	            IF #Transf.Dial_Def.Reponse_Def = 'Cellule' AND #Transf.Dial_Def.Num_Def_Etape = 1 THEN // cellule
	                #Ret_Int := "Index_Mobile"(#Transf.Dial_Def.Text_Reponse);
	                #Transf.Dial_Def.Reponse_Def := '';
	                IF #Ret_Int <= -1 THEN
	                    #Text_Def := CONCAT(IN1 := 'Cellule ', IN2 := #Transf.Dial_Def.Text_Reponse, IN3 := ' Inexistante');
	                    #Transf.Dial_Def.Index_Defaut := "Dialog_Defaut"(Fg_Base := #fgbase, Msg_Defaut := #Text_Def,
	                                                                     Type_Defaut := 2,
	                                                                     Automatisme := #Transf._TransfCommun.CommunGeneral._Autom,
	                                                                     Num_Lot := #Transf._PtCir.Num_Lot,
	                                                                     Origine_Defaut := #Text_Def,
	                                                                     Libelle_Origine := 'Cellule inexistante',
	                                                                     Acq1 := 'Relance',
	                                                                     Acq2 := 'Cellule',
	                                                                     Acq3 := '',
	                                                                     Acq4 := '',
	                                                                     Acq5 := '',
	                                                                     Acq6 := '',
	                                                                     Acq7 := '',
	                                                                     Acq8 := '',
	                                                                     Acq_Choisi := -1,
	                                                                     Date_Arrivee := #Transf._TpsPicke);
	                    #Transf._TransfCommun.CommunGeneral._Etp := #Etape_Attente_RepDial;
	                    #Transf.Dial_Def.Text_Reponse := '';
	                    RETURN;
	                ELSE
	                    #Transf._CelluleTrouve := "Controle_Cellule"(FgMaskNh := #Transf._FgMaskCtrlNh,
	                                                                 NvCellule := #Transf.Dial_Def.Text_Reponse,
	                                                                 TypeCelDest := #Transf._TypeCelDest,
	                                                                 Cel := "DB_Mod_Cellule",
	                                                                 NiveauHautDestNh => #Transf._NiveauHautDestNh);
	                END_IF;
	            END_IF;
	            //============ fIN Traitement des reponses pour le defaut1 Etape CHANGEMENT DE DESTINATION cellule introuvable  ===============================//






	            ////Test invalide de la destination recuperee de la Base, cellule est en nh
	            IF #Transf._CelluleTrouve = 1 THEN
	                #Transf.Dial_Def.Num_Def_Etape := 2;
	                #Text_Def := CONCAT(IN1 := 'Cellule ', IN2 := #Transf.Dial_Def.Text_Reponse, IN3 := '  est en NH');
	                #Transf.Dial_Def.Index_Defaut := "Dialog_Defaut"(Fg_Base := #fgbase, Msg_Defaut := #Text_Def,
	                                                                 Type_Defaut := 2,
	                                                                 Automatisme := #Transf._TransfCommun.CommunGeneral._Autom,
	                                                                 Num_Lot := #Transf._Ptzs._NoLot,
	                                                                 Origine_Defaut := #Text_Def,
	                                                                 Libelle_Origine := #Text_Def,
	                                                                 Acq1 := 'Relance',
	                                                                 Acq2 := 'Cellule',
	                                                                 Acq3 := '', //'Forçage'
	                                                                 Acq4 := '',
	                                                                 Acq5 := '',
	                                                                 Acq6 := '',
	                                                                 Acq7 := '',
	                                                                 Acq8 := '',
	                                                                 Acq_Choisi := -1,
	                                                                 Date_Arrivee := #Transf._TpsPicke);
	                #Transf._TransfCommun.CommunGeneral._Etp := #Etape_Attente_RepDial;
	                RETURN;
	            END_IF;
	        CHANGEMENT_DEST_DEF2:
	            //============ Traitement des reponses pour le defaut2 Etape CHANGEMENT DE DESTINATION cellule en nh  ====================================//
	            IF #Transf.Dial_Def.Reponse_Def = 'Relance' AND #Transf.Dial_Def.Num_Def_Etape = 2 THEN
	                #Transf._CelluleTrouve := "Controle_Cellule"(FgMaskNh := #Transf._FgMaskCtrlNh,
	                                                             NvCellule := #Transf.Dial_Def.Text_Reponse,
	                                                             TypeCelDest := #Transf._TypeCelDest,
	                                                             Cel := "DB_Mod_Cellule",
	                                                             NiveauHautDestNh => #Transf._NiveauHautDestNh);
	                #Transf.Dial_Def.Text_Reponse := '';
	                RETURN;
	            END_IF;


	            IF #Transf.Dial_Def.Reponse_Def = 'Forcage' AND #Transf.Dial_Def.Num_Def_Etape = 2 THEN
	                #Transf._FgMaskCtrlNh := TRUE;
	                #Transf._FgChangDest := FALSE;
	                #Transf._TransfCommun.SUPTRANS.Commande._FgChangDest := FALSE;
	                #Transf._Ptzs._DestR._Liste[#Transf._Ptzs._DestR._Index]._Nh := FALSE;
	                #Transf._CelluleTrouve := 2;
	                #Transf._TransfCommun.CommunGeneral._Ptdest := "Index_Mobile"(#Transf.Dial_Def.Text_Reponse);
	                #Transf._IndexDestEc := "RechIndexCel"("Nom_Mobile"(#Transf._TransfCommun.CommunGeneral._Ptdest));
	                IF #Transf._IndexDestEc > -1 THEN
	                    #Transf._ptDestEc := "DB_Mod_Cellule"._TabCel[#Transf._IndexDestEc];
	                END_IF;
	                (* "MAJ_Cumul_Dest"(Dest := "Nom_Mobile"(#Transf.TransfCommun.CommunGeneral._Ptdest),
	                                  Increment := FALSE,
	                                  DestR := #Transf._Ptzs._DestR,
	                                  PARCAL := #Transf.TransfCommun.CommunGeneral._ParCal);
	                 #Transf._CumulQteNh := #Transf._Ptzs._DestR._Liste[#Transf._Ptzs._DestR._Index]._CumulQte;
	                 (* #Transf.transfCommun.CommunGeneral._Ptdest := "Index_Mobile"(#Transf.Dial_Def.Text_Reponse);
	                 #Transf._IndexDestEc := "RechIndexCel"("Nom_Mobile"(#Transf.transfCommun.CommunGeneral._Ptdest)); *)
	                "ChngDestNoeud_Transfert"(#Transf); *)
	                #Transf.Dial_Def.Reponse_Def := '';
	            END_IF;



	            IF #Transf.Dial_Def.Reponse_Def = 'Cellule' AND #Transf.Dial_Def.Num_Def_Etape = 2 THEN // cellule
	                #Ret_Int := "Index_Mobile"(#Transf.Dial_Def.Text_Reponse);
	                #Transf.Dial_Def.Reponse_Def := '';
	                IF #Ret_Int <= -1 THEN
	                    #Transf._CelluleTrouve := 0;
	                    #Transf.Dial_Def.Num_Def_Etape := 1;
	                    #Text_Def := CONCAT(IN1 := 'Cellule ', IN2 := #Transf.Dial_Def.Text_Reponse, IN3 := '  inexistante');
	                    #Transf.Dial_Def.Index_Defaut := "Dialog_Defaut"(Fg_Base := #fgbase, Msg_Defaut := #Text_Def,
	                                                                     Type_Defaut := 2,
	                                                                     Automatisme := #Transf._TransfCommun.CommunGeneral._Autom,
	                                                                     Num_Lot := #Transf._PtCir.Num_Lot,
	                                                                     Origine_Defaut := 'Cellule inexistante',
	                                                                     Libelle_Origine := 'Cellule inexistante',
	                                                                     Acq1 := 'Relance',
	                                                                     Acq2 := 'Cellule',
	                                                                     Acq3 := '',
	                                                                     Acq4 := '',
	                                                                     Acq5 := '',
	                                                                     Acq6 := '',
	                                                                     Acq7 := '',
	                                                                     Acq8 := '',
	                                                                     Acq_Choisi := -1,
	                                                                     Date_Arrivee := #Transf._TpsPicke);
	                    #Transf._TransfCommun.CommunGeneral._Etp := #Etape_Attente_RepDial;
	                    #Transf.Dial_Def.Text_Reponse := '';
	                    RETURN;
	                ELSE
	                    #Transf._CelluleTrouve := "Controle_Cellule"(FgMaskNh := #Transf._FgMaskCtrlNh,
	                                                                 NvCellule := #Transf.Dial_Def.Text_Reponse,
	                                                                 TypeCelDest := #Transf._TypeCelDest,
	                                                                 Cel := "DB_Mod_Cellule",
	                                                                 NiveauHautDestNh => #Transf._NiveauHautDestNh);
	                END_IF;
	            END_IF;

	            //============ FIN Traitement des reponses pour le defaut2 Etape CHANGEMENT DE DESTINATION cellule en nh  ====================================//



	            IF #Transf._CelluleTrouve = 3 THEN // CELLULE RECUP VALID MAIS LA RECHERCHERCHE DU NV CIRC RETURN-1
	                #Transf.Dial_Def.Num_Def_Etape := 1;
	                #Text_Def := CONCAT(IN1 := 'Circuit de ', IN2 := "Nom_Mobile"(#Transf._TransfCommun.CommunGeneral._PtOrig), IN3 := ' vers ', IN4 := #Transf.Dial_Def.Text_Reponse, IN5 := ' introuvable ou reserve ');
	                #Transf.Dial_Def.Index_Defaut := "Dialog_Defaut"(Fg_Base := #fgbase, Msg_Defaut := #Text_Def,
	                                                                 Type_Defaut := 2,
	                                                                 Automatisme := #Transf._TransfCommun.CommunGeneral._Autom,
	                                                                 Num_Lot := #Transf._Ptzs._NoLot,
	                                                                 Origine_Defaut := 'Circuit Introuvable',
	                                                                 Libelle_Origine := 'Circuit Introuvable',
	                                                                 Acq1 := 'Relance',
	                                                                 Acq2 := 'Cellule',
	                                                                 Acq3 := '',
	                                                                 Acq4 := '',
	                                                                 Acq5 := '',
	                                                                 Acq6 := '',
	                                                                 Acq7 := '',
	                                                                 Acq8 := '',
	                                                                 Acq_Choisi := -1,
	                                                                 Date_Arrivee := #Transf._TpsPicke);
	                #Transf._TransfCommun.CommunGeneral._Etp := #Etape_Attente_RepDial;
	                RETURN;
	            END_IF;


	            //Test valide de la destination recuperee
	            IF #Transf._CelluleTrouve = 2 THEN
	                IF #Transf._TransfCommun.CommunGeneral._IndxDest <> #ListeDestParcourue THEN
	                    #CdZoneDest := "Nom_Mobile"(#Transf._TransfCommun.CommunGeneral._Dest[#Transf._TransfCommun.CommunGeneral._IndxDest]);
	                ELSE
	                    #CdZoneDest := #Transf.Dial_Def.Text_Reponse;
	                END_IF;
	                #Anc_Dest := "Nom_Mobile"(#Transf._TransfCommun.CommunGeneral._AncDest);
	                (* "ControleDestTransf"(fgbase := fgbase,
	                                     "Return" => #Ret_Int,
	                                     Transf := #Transf,
	                                     NoLot := #Transf._Ptzs._NoLot,
	                                     CdZoneDest := #CdZoneDest,
	                                     Anc_Dest := #Anc_Dest,
	                                     Nouv_Dest := #Transf._Ptzs._NouvDest,
	                                     CdMat := #Transf._Ptzs._CdMat,
	                                     NomAuto := #Transf.TransfCommun.CommunGeneral._Autom); *)

	                "ControleDest"(fgbase := #fgbase,
	                               TypeCelDest := #Transf._TypeCelDest,
	                               FgMaskCtrlNh := #Transf._FgMaskCtrlNh,
	                               "Return" => #Ret_Int,
	                               FgLanc => #Transf._FgLanc,
	                               NiveauHautDestNh => #Transf._NiveauHautDestNh,
	                               CntlDest := #Transf.CntlDest,
	                               Dial_Def := #Transf.Dial_Def,
	                               NoLot := #Transf._Ptzs._NoLot,
	                               CdZoneDest := #CdZoneDest,
	                               Anc_Dest := #Anc_Dest,
	                               Nouv_Dest := #Transf._Ptzs._NouvDest,
	                               CdMat := #Transf._Ptzs._CdMat,
	                               NomAuto := #Transf._TransfCommun.CommunGeneral._Autom);

	                IF #Ret_Int = -1 THEN
	                    #Transf._CelluleTrouve := 0;
	                END_IF;
	                IF #Ret_Int = 1 THEN
	                    #Transf._CumulQteNh := #Transf._Ptzs._DestR._Liste[#Transf._Ptzs._DestR._Index]._CumulQte;
	                    // IF #Transf.TransfCommun.CommunGeneral._IndxDest <= "NB_MAX_DEST" THEN //AND #Transf.Dial_Def.Num_Def_Etape = 0 THEN
	                    IF #Transf._TransfCommun.CommunGeneral._IndxDest <> #ListeDestParcourue THEN
	                        #Transf._TransfCommun.CommunGeneral._Ptdest := #Transf._TransfCommun.CommunGeneral._Dest[#Transf._TransfCommun.CommunGeneral._IndxDest];
	                    ELSE
	                        #Transf._TransfCommun.CommunGeneral._Ptdest := "Index_Mobile"(#Transf.Dial_Def.Text_Reponse);
	                    END_IF;
	                    #Transf._IndexDestEc := "RechIndexCel"("Nom_Mobile"(#Transf.#_TransfCommun.CommunGeneral._Ptdest));
	                    IF #Transf._IndexDestEc > -1 THEN
	                        #Transf._ptDestEc := "DB_Mod_Cellule"._TabCel[#Transf._IndexDestEc];
	                    END_IF;
	                    #Transf._TransfCommun.CommunGeneral._Etp := #Etape_ChgmtDestNoeud;
	                    RETURN;

	                END_IF;


	                (* #Transf._CumulQteNh := #Transf._Ptzs._DestR._Liste[#Transf._Ptzs._DestR._Index]._CumulQte;
	                 // IF #Transf.TransfCommun.CommunGeneral._IndxDest <= "NB_MAX_DEST" THEN //AND #Transf.Dial_Def.Num_Def_Etape = 0 THEN
	                 IF #Transf.TransfCommun.CommunGeneral._IndxDest <> #ListeDestParcourue THEN
	                     #Transf.TransfCommun.CommunGeneral._Ptdest := #Transf.TransfCommun.CommunGeneral._Dest[#Transf.TransfCommun.CommunGeneral._IndxDest];
	                 ELSE
	                     #Transf.TransfCommun.CommunGeneral._Ptdest := "Index_Mobile"(#Transf.Dial_Def.Text_Reponse);
	                 END_IF;
	                 #Transf._IndexDestEc := "RechIndexCel"("Nom_Mobile"(#Transf.#TransfCommun.CommunGeneral._Ptdest));
	                 IF #Transf._IndexDestEc > -1 THEN
	                     #Transf._ptDestEc := "DB_Mod_Cellule"._TabCel[#Transf._IndexDestEc];
	                 END_IF;
	                 "ChngDestNoeud_Transfert"(#Transf); *)
	            END_IF;







	            (* IF #Transf.TransfCommun.CommunGeneral._IndxDest <> #ListeDestParcourue THEN
	                 #CdZoneDest := "Nom_Mobile"(#Transf.TransfCommun.CommunGeneral._Dest[#Transf.TransfCommun.CommunGeneral._IndxDest]);
	             ELSE
	                 #CdZoneDest := #Transf.Dial_Def.Text_Reponse;
	             END_IF;
	             #Anc_Dest := "Nom_Mobile"(#Transf.TransfCommun.CommunGeneral._AncDest);
	             "ControleDestTransf"(fgbase:=fgbase,
	                                  "Return"=>#Ret_Int,
	                                  Transf:=#Transf,
	                                  NoLot:=#Transf._Ptzs._NoLot,
	                                  CdZoneDest:= #CdZoneDest,
	                                  Anc_Dest:= #Anc_Dest,
	                                  Nouv_Dest:=#Transf._Ptzs._NouvDest,
	                                  CdMat:=#Transf._Ptzs._CdMat,
	                                  NomAuto:=#Transf.TransfCommun.CommunGeneral._Autom);
	             IF #Ret_Int =1 THEN
	                 #Transf._CelluleTrouve := 2 ;
	             ELSE
	                 #Transf._CelluleTrouve := -2;
	             END_IF; *)

	        END_REGION Traitement cyclique
	(*
	 *************************************** *************************************** *************************************** *************************************** *************************************** ***************************************
	                                                                                 ╔════════════════════════════════════╗
	                                                                                 ║          ChgmtDestNoeud            ║
	                                                                                 ╚════════════════════════════════════╝
	 *************************************** *************************************** *************************************** *************************************** *************************************** ***************************************
	*)
	    #Etape_ChgmtDestNoeud:
	        REGION Traitement preliminaire 'ChgmtDestNoeud'
	            IF (#Transf._TransfCommun.CommunGeneral._Etp <> #Transf._TransfCommun.CommunGeneral._EtpPrec) THEN
	                //Memorisation de l'etape encours
	                #Transf._TransfCommun.CommunGeneral._EtpPrec := #Transf._TransfCommun.CommunGeneral._Etp;
	                //Reperer le niveau du grafcet
	                #MajNiv := "Maj_Niv"(Num_Zone := #Transf._TransfCommun.CommunGeneral._NumZone, Num_Tache := #Transf._TransfCommun.CommunGeneral._Tache, Niveau := "TRANSF_ChangementNoeud_Niv");
	                //Nomination l'etape en cours
	                #Transf._TransfCommun.CommunGeneral._DescEtp := 'Etape ChgmtDestNoeud';
	                //lecture du temps local
	                #Ret_RD_Sys_T := RD_SYS_T(#Transf._TpsPicke);
	                IF #Transf.Dial_Def.Reponse_Def <> '' THEN
	                    CASE #Transf.Dial_Def.Num_Def_Etape OF
	                        1:
	                            GOTO ProcChangDest_DEF1;
	                    END_CASE;
	                END_IF;
	            END_IF;
	        END_REGION Traitement preliminaire 'ChgmtDestNoeud'
	        REGION Traitement cyclique 'ChgmtDestNoeud'
	            #ReturnChngDest := "ChngDest"(NouvDest := #Transf._TransfCommun.CommunGeneral._Ptdest,
	                                          AncDest := #Transf._TransfCommun.CommunGeneral._AncDest,
	                                          IndxDestEncours := #Transf._TransfCommun.CommunGeneral._IndxDest,
	                                          ChNoeud := #Transf.ChNoeud,
	                                          AncCircuit := #Transf._PtCir,
	                                          CelluleTrouve := #Transf._CelluleTrouve,
	                                          FgChangementDest := #Transf._FgChangDest);
	            IF #ReturnChngDest = -3 THEN //rech circ return -1 et
	                #Transf._CelluleTrouve := 3;
	                #Transf._TransfCommun.CommunGeneral._Etp := #Etape_changement_destination;
	                RETURN;
	            END_IF;
	            IF #ReturnChngDest = -2 THEN //rech circ return -1
	                #Transf._CelluleTrouve := 0;
	                #Transf._TransfCommun.CommunGeneral._Etp := #Etape_changement_destination;
	                RETURN;
	            END_IF;
	            IF #ReturnChngDest = 1 THEN // valide
	                IF #fgbase THEN
	                    IF #Transf._Ptzs._DestR._Index > 1 THEN
	                        #ResultProcChangmtdesttransf := "Proc_Changement_Dest_TRANSF"(NumPoste := "Num_Poste", IdTransf := #Transf._Ptzs._Id_Transf,
	                                                                                      AncDest := "Nom_Mobile"(#Transf._TransfCommun.CommunGeneral._AncDest),
	                                                                                      NvDest := "Nom_Mobile"(#Transf._TransfCommun.CommunGeneral._Ptdest),
	                                                                                      QTE := #Transf._Ptzs._DestR._Liste[#Transf._Ptzs._DestR._Index - 1]._Qte,
	                                                                                      TpsMarche := #Transf._Ptzs._DestR._Liste[#Transf._Ptzs._DestR._Index - 1]._Tps / 1000,
	                                                                                      MajStock := 'R', Msg_Def => #Text_Def);
	                    ELSE
	                        #ResultProcChangmtdesttransf := "Proc_Changement_Dest_TRANSF"(NumPoste := "Num_Poste", IdTransf := #Transf._Ptzs._Id_Transf,
	                                                                                      AncDest := "Nom_Mobile"(#Transf._TransfCommun.CommunGeneral._AncDest),
	                                                                                      NvDest := "Nom_Mobile"(#Transf._TransfCommun.CommunGeneral._Ptdest),
	                                                                                      QTE := #Transf._TransfCommun.CommunGeneral._ParCal._QteTrans,
	                                                                                      TpsMarche := #Transf._TransfCommun.CommunGeneral._ParCal._TpsTran / 1000,
	                                                                                      MajStock := 'R', Msg_Def => #Text_Def);
	                    END_IF;
	                ELSE
	                    #ResultProcChangmtdesttransf := 'OK';
	                END_IF;



	                IF #ResultProcChangmtdesttransf = 'OK' THEN
	                    #ret_string := "Proc_AffecT"(NumPoste := "Num_Poste",
	                                                 zone := "Nom_Mobile"(#Transf._TransfCommun.CommunGeneral._Ptdest),
	                                                 CodeMat := #Transf._Ptzs._CdMat,
	                                                 Formule := #Temp_Char,
	                                                 LieuDos := '',
	                                                 Qte := 0,
	                                                 TypeMvmnt := '040',
	                                                 Procede := #Transf._TransfCommun.CommunGeneral._Autom,
	                                                 NoLotOrig := '',
	                                                 NoLotDest := #Transf._Ptzs._NoLot,
	                                                 Utilisateur := 'SAS',
	                                                 SCb := '0',
	                                                 Sof := #Transf._Ptzs._Cd_Transf, Msg_Def => #Text_Def);
	                    #Transf.Dial_Def.Reponse_Def := '';
	                    #Transf.Dial_Def.Text_Reponse := '';
	                    #Transf._CelluleTrouve := 0;
	                    #Transf._FgChangDest := FALSE;
	                    #Transf._TransfCommun.SUPTRANS.Commande._FgChangDest := FALSE;
	                    IF #Transf._Ptzs._Fg_Produit_Vu = TRUE THEN
	                        #Transf._TransfCommun.CommunGeneral._Etp := #Etape_surveillance;
	                    ELSE
	                        #Transf._TransfCommun.CommunGeneral._Etp := #Etape_attente_produit;
	                    END_IF;
	                    RETURN;
	                END_IF;
	                IF #ResultProcChangmtdesttransf = 'NOK' THEN
	                    #Transf.Dial_Def.Num_Def_Etape := 1;
	                    #Transf.Dial_Def.Index_Defaut := "Dialog_Defaut"(Fg_Base := #fgbase, Msg_Defaut := #Text_Def,
	                                                                     Type_Defaut := 2,
	                                                                     Automatisme := #Transf._TransfCommun.CommunGeneral._Autom,
	                                                                     Num_Lot := #Transf._Ptzs._NoLot,
	                                                                     Origine_Defaut := 'Base de donnees',
	                                                                     Libelle_Origine := 'Base de donnees',
	                                                                     Acq1 := 'Abandon',
	                                                                     Acq2 := 'Relance',
	                                                                     Acq3 := '',
	                                                                     Acq4 := '',
	                                                                     Acq5 := '',
	                                                                     Acq6 := '',
	                                                                     Acq7 := '',
	                                                                     Acq8 := '',
	                                                                     Acq_Choisi := -1,
	                                                                     Date_Arrivee := #Transf._TpsPicke);
	                    #Transf._TransfCommun.CommunGeneral._Etp := #Etape_Attente_RepDial;
	                    RETURN;
	                END_IF;
	            END_IF;
	        ProcChangDest_DEF1:
	            //============ Traitement des reponses pour le defaut1   Traitement_Badge=============================================================//
	            IF #Transf.Dial_Def.Reponse_Def = 'Relance' THEN
	                #Transf.Dial_Def.Reponse_Def := '';
	                #Transf._TransfCommun.CommunGeneral._Etp := #Etape_ChgmtDestNoeud;
	                RETURN;
	            END_IF;
	            IF #Transf.Dial_Def.Reponse_Def = 'Abandon' THEN
	                IF #Transf._Ptzs._Fg_Produit_Vu = TRUE THEN
	                    #Transf._TransfCommun.CommunGeneral._Etp := #Etape_surveillance;
	                ELSE
	                    #Transf._TransfCommun.CommunGeneral._Etp := #Etape_attente_produit;
	                END_IF;
	                #Transf.Dial_Def.Reponse_Def := '';
	                RETURN;
	            END_IF;
	            //============================================  Fin traitement  ====================================================================//





	        END_REGION Traitement cyclique

	(*
	 *************************************** *************************************** *************************************** *************************************** *************************************** ***************************************
	                                                                                 ╔════════════════════════════════════╗
	                                                                                 ║      Etape Changement origine      ║
	                                                                                 ╚════════════════════════════════════╝
	 *************************************** *************************************** *************************************** *************************************** *************************************** ***************************************
	*)


	(*
	 *************************************** *************************************** *************************************** *************************************** *************************************** ***************************************
	                                                                                 ╔════════════════════════════════════╗
	                                                                                 ║           Etape Vidange            ║
	                                                                                 ╚════════════════════════════════════╝
	 *************************************** *************************************** *************************************** *************************************** *************************************** ***************************************
	*)
	    #Etape_vidange:
	        REGION Traitement preliminaire 'Vidange'

	            IF (#Transf._TransfCommun.CommunGeneral._Etp <> #Transf._TransfCommun.CommunGeneral._EtpPrec) THEN
	                //Memorisation de l'etape encours
	                #Transf._TransfCommun.CommunGeneral._EtpPrec := #Transf._TransfCommun.CommunGeneral._Etp;
	                //Reperer le niveau du grafcet
	                #MajNiv := "Maj_Niv"(Num_Zone := #Transf._TransfCommun.CommunGeneral._NumZone, Num_Tache := #Transf._TransfCommun.CommunGeneral._Tache, Niveau := "TRANSF_Vidange_Niv");
	                //Nomination l'etape en cours
	                #Transf._TransfCommun.CommunGeneral._DescEtp := 'Etape Vidange';
	                // Memorise la quantit au dmarrage de la vidnage
	                IF #Transf._Ptzs._ArretReel = 'Quantite' AND #Transf._FgColChute THEN
	                    #Transf._QteAvVid := #Transf._TransfCommun.CommunGeneral._ParCal._QteTrans;
	                END_IF;
	                IF #Transf._FgValidMvmtSortie AND #Transf._Ptzs._ArretReel = 'Niveau bas' THEN
	                    ///
	                    //
	                    ;
	                END_IF;
	                (* #Ret_Int := "RechIndexCel"("Nom_Mobile"("Index_Mobile"(#Transf._orig.Nom)));
	               "Arret_Ext_Libere"(Origine := "DB_Mod_Cellule"._TabCel[#Ret_Int]); *)
	                #Ret_Int := "RechIndexCel"("Nom_Mobile"(#Transf._TransfCommun.CommunGeneral._PtOrig));
	                // "Arret_Ext_Libere"(Origine := "DB_Mod_Cellule"._TabCel[#Ret_Int]);
	                "MarcheExt"(Origine := #Transf._TransfCommun.CommunGeneral._PtOrig,
	                            Position := #PosFerm,
	                            Vitesse := 0);

	                #Transf._FgDemVid := FALSE;


	                #Transf._Ptzs._QteLot := #Transf._TransfCommun.CommunGeneral._ParCal._QteTrans;

	                // #Ret_Int := "Fin_Pos_Circuit"(#Transf._PtCir);
	            END_IF;
	        END_REGION Traitement preliminaire 'Vidange'

	        REGION Traitement cyclique "Vidange"
	            #Ret_Bool := "Vid_Circuit_Cycl"(#Transf._PtCir);
	            IF #Ret_Bool AND "Test_Etat_Circuit"(Etat := "Libre", Debut := 0, CIRCUIT := #Transf._PtCir) THEN
	                //IF "Test_Etat_Circuit"(Etat := "Enc_Fin_Pos", Debut := 0, CIRCUIT := #Transf._PtCir) THEN
	                #Ret_Int := "Libere_Circuit"(#Transf._PtCir);
	                // Mise a jour de la colonne de chute
	                IF #Transf._Ptzs._ArretReel = 'Quantite' AND #Transf._FgColChute THEN
	                    #Transf._colChute := (#Transf._TransfCommun.CommunGeneral._ParCal._QteTrans - #Transf._QteAvVid);
	                    IF #Transf._colChute > (#Transf._Ptzs._Colchute + #Transf._corColChute) AND #Transf._Ptzs._Colchute <> 0 THEN
	                        #Transf._colChute := #Transf._Ptzs._Colchute + #Transf._corColChute;
	                    ELSIF #Transf._colChute < (#Transf._Ptzs._Colchute + #Transf._corColChute) AND #Transf._Ptzs._Colchute <> 0 THEN
	                        #Transf._colChute := #Transf._Ptzs._Colchute - #Transf._corColChute;
	                    END_IF;
	                    // appel Proc_MajColChute(pt_zs->OrigReel,_colChute);
	                END_IF;
	                "MAJ_Cumul_Dest"(Dest := "Nom_Mobile"(#Transf._TransfCommun.CommunGeneral._Ptdest),
	                                 Increment := FALSE,
	                                 DestR := #Transf._Ptzs._DestR,
	                                 PARCAL := #Transf._TransfCommun.CommunGeneral._ParCal);


	                #Transf._CumulQteNh := #Transf._Ptzs._DestR._Liste[#Transf._Ptzs._DestR._Index]._CumulQte;
	                #Transf._TransfCommun.CommunGeneral._Etp := #Etape_MAJ_Base;
	            END_IF;
	        END_REGION Traitement cyclique "Vidange"


	        RETURN;

	(*
	 *************************************** *************************************** *************************************** *************************************** *************************************** ***************************************
	                                                                                 ╔════════════════════════════════════╗
	                                                                                 ║           Etape MAJ Base           ║
	                                                                                 ╚════════════════════════════════════╝
	 *************************************** *************************************** *************************************** *************************************** *************************************** ***************************************
	*)
	    #Etape_MAJ_Base:
	        REGION Traitement preliminaire 'Maj Base'
	            IF (#Transf._TransfCommun.CommunGeneral._Etp <> #Transf._TransfCommun.CommunGeneral._EtpPrec) THEN
	                //Memorisation de l'etape encours
	                #Transf._TransfCommun.CommunGeneral._EtpPrec := #Transf._TransfCommun.CommunGeneral._Etp;
	                //Reperer le niveau du grafcet

	                #MajNiv := "Maj_Niv"(Num_Zone := #Transf._TransfCommun.CommunGeneral._NumZone, Num_Tache := #Transf._TransfCommun.CommunGeneral._Tache, Niveau := "TRANSF_MajBase_Niv");
	                //Nomination l'etape en cours
	                #Transf._TransfCommun.CommunGeneral._DescEtp := 'Maj Base';
	            END_IF;
	        END_REGION Traitement preliminaire 'Maj Base'

	        REGION Traitement cyclique "Maj Base"
	            IF #Transf._FgGestDens THEN
	                #ret_sint := "CorDensite"(QteReelle := #Transf._Ptzs._QtePrev,
	                                          QteCalculee := #Transf._TransfCommun.CommunGeneral._ParCal._QteTrans,
	                                          AncCoeff := #Transf._Ptzs._CoefDens,
	                                          PasMaxCorCoeff := #Transf._PasMaxCorCoeff,
	                                          DensCorMax := #Transf._DensMaxi,
	                                          DensCorMin := #Transf._DensMini,
	                                          DensInitial := #Transf._Ptzs._Densite,
	                                          TolMax := #Transf._TolMax,
	                                          TolMin := #Transf._TolMin,
	                                          NvCoeff := #Transf._AffCoefCor,
	                                          DensCor := #Transf._AffDensCours);
	            END_IF;
	            IF #fgbase AND #ret_sint = 0 THEN
	                // Appel Proc RecrCoef Proc_RecrCoef(pt_zs->Cd_Mat,LireIdIdCoeffDens(),AnsiString(WLireProcede()).c_str(),_nouvCoef);
	                ;
	            END_IF;




	            //*Maj_Etape(_ta, "fin_lot");
	            #Transf._TransfCommun.CommunGeneral._Etp := #Etape_Fin_Lot;
	        END_REGION Traitement cyclique "Maj Base"
	        RETURN;


	(*
	 *************************************** *************************************** *************************************** *************************************** *************************************** ***************************************
	                                                                                 ╔════════════════════════════════════╗
	                                                                                 ║           Etape Fin Lot            ║
	                                                                                 ╚════════════════════════════════════╝
	 *************************************** *************************************** *************************************** *************************************** *************************************** ***************************************
	*)
	    #Etape_Fin_Lot:
	        REGION Traitement preliminaire 'Fin Lot'
	            IF (#Transf._TransfCommun.CommunGeneral._Etp <> #Transf._TransfCommun.CommunGeneral._EtpPrec) THEN
	                //Memorisation de l'etape encours
	                #Transf._TransfCommun.CommunGeneral._EtpPrec := #Transf._TransfCommun.CommunGeneral._Etp;
	                //Nomination l'etape en cours
	                #Transf._TransfCommun.CommunGeneral._DescEtp := 'Fin Lot';
	                #Transf._FgArret := FALSE;
	                IF #Transf.Dial_Def.Reponse_Def <> '' THEN
	                    CASE #Transf.Dial_Def.Num_Def_Etape OF
	                        1:
	                            GOTO FinLot_DEF1;
	                    END_CASE;
	                END_IF;
	                IF #fgbase THEN
	                    #ResultProcFintransf := "Proc_Fin_Transf"(IdTransf := #Transf._Ptzs._Id_Transf,
	                                                              CumulTps := #Transf._TransfCommun.CommunGeneral._ParCal._TpsTran / 1000,
	                                                              CumulQte := #Transf._TransfCommun.CommunGeneral._ParCal._QteTrans,
	                                                              CModArr := #Transf._Ptzs._TypeArret,
	                                                              NumPoste := "Num_Poste", Msg_Def => #Text_Def);
	                ELSE
	                    #ResultProcFintransf := 'OK';
	                END_IF;


	            END_IF;
	        END_REGION Traitement preliminaire 'Fin Lot'

	        REGION Traitement cyclique "Fin Lot"
	            IF #ResultProcFintransf = 'NOK' THEN
	                #Transf.Dial_Def.Num_Def_Etape := 1;
	                #Transf.Dial_Def.Index_Defaut := "Dialog_Defaut"(Fg_Base := #fgbase, Msg_Defaut := #Text_Def,
	                                                                 Type_Defaut := 2,
	                                                                 Automatisme := #Transf._TransfCommun.CommunGeneral._Autom,
	                                                                 Num_Lot := #Transf._Ptzs._NoLot,
	                                                                 Origine_Defaut := 'Base de donnees',
	                                                                 Libelle_Origine := 'Base de donnees',
	                                                                 Acq1 := 'Abandon',
	                                                                 Acq2 := 'Relance',
	                                                                 Acq3 := '',
	                                                                 Acq4 := '',
	                                                                 Acq5 := '',
	                                                                 Acq6 := '',
	                                                                 Acq7 := '',
	                                                                 Acq8 := '',
	                                                                 Acq_Choisi := -1,
	                                                                 Date_Arrivee := #Transf._TpsPicke);
	                #Transf._TransfCommun.CommunGeneral._Etp := #Etape_Attente_RepDial;
	                RETURN;
	            END_IF;
	        FinLot_DEF1:
	            //================================== Traitement des reponses pour le defaut1  =============================================================//
	            IF #Transf.Dial_Def.Reponse_Def = 'Abandon' THEN
	                #ResultProcFintransf := 'OK';
	                #Transf.Dial_Def.Reponse_Def := '';
	            END_IF;
	            IF #Transf.Dial_Def.Reponse_Def = 'Relance' THEN
	                #Transf.Dial_Def.Reponse_Def := '';
	                #ResultProcFintransf := "Proc_Fin_Transf"(IdTransf := #Transf._Ptzs._Id_Transf,
	                                                          CumulTps := #Transf._TransfCommun.CommunGeneral._ParCal._TpsTran / 1000,
	                                                          CumulQte := #Transf._TransfCommun.CommunGeneral._ParCal._QteTrans,
	                                                          CModArr := #Transf._Ptzs._TypeArret,
	                                                          NumPoste := "Num_Poste", Msg_Def => #Text_Def);
	            END_IF;
	            //============================================  Fin traitement  ====================================================================//
	            IF #ResultProcFintransf = 'OK' THEN
	                #MajNiv := "Maj_Niv"(Num_Zone := #Transf._TransfCommun.CommunGeneral._NumZone, Num_Tache := #Transf._TransfCommun.CommunGeneral._Tache, Niveau := "TRANSF_FinLot_Niv");
	                #Ret_Int := "Libere_Zone_Suiv_Lot"(Num_Zone := #Transf._TransfCommun.CommunGeneral._NumZone);
	                #Transf._TransfCommun.SUPTRANS.Commande._Suspension := FALSE;
	                #Transf._TransfCommun.SUPTRANS.Commande._Vidange := FALSE;
	                #Transf._TransfCommun.SUPTRANS.Commande._ArretImmediat := FALSE;
	                #Transf._TransfCommun.SUPTRANS.Commande._Depart := FALSE;
	                "Supervision_Transf"(RAZ := TRUE,
	                                     Transf := #Transf);
	                //#Transf.TraitTransf.Etape := 0;
	                #Transf._TransfCommun.CommunGeneral._Etp := #Etape_Repos;
	                RETURN;
	            END_IF;

	        END_REGION Traitement cyclique "Fin Lot"
	        RETURN;



	(*
	 *************************************** *************************************** *************************************** *************************************** *************************************** ***************************************
	                                                                                 ╔════════════════════════════════════╗
	                                                                                 ║       Etape test ench orig         ║
	                                                                                 ╚════════════════════════════════════╝
	 *************************************** *************************************** *************************************** *************************************** *************************************** ***************************************
	*)














	(*
	 *************************************** *************************************** *************************************** *************************************** *************************************** ***************************************
	                                                                                 ╔════════════════════════════════════╗
	                                                                                 ║ Etape "Attente Reponse Dialogue"   ║
	                                                                                 ╚════════════════════════════════════╝
	 *************************************** *************************************** *************************************** *************************************** *************************************** ***************************************
	*)
	    #Etape_Attente_RepDial:
	        REGION Preliminaire Attente Acquuitement
	            IF #Transf._TransfCommun.CommunGeneral._Etp <> #Transf._TransfCommun.CommunGeneral._EtpPrec THEN
	                //Memorisation de l'etape encours
	                #Transf._TransfCommun.CommunGeneral._EtpMemo := #Transf._TransfCommun.CommunGeneral._EtpPrec;

	                #Transf._TransfCommun.CommunGeneral._DescEtp := 'Etape_Attente_RepDial';
	                #Transf._TransfCommun.CommunGeneral._EtpPrec := #Transf._TransfCommun.CommunGeneral._Etp;

	            END_IF;
	        END_REGION Preliminaire Attente Acquuitement
	        REGION Cyclique Attente Acquitement
	            #Transf.Dial_Def.Reponse_Def := "FC_Recup_Rep_Def"(Index_Def := #Transf.Dial_Def.Index_Defaut, Reponse_Ecrit => #Transf.Dial_Def.Text_Reponse);
	            IF #Transf.Dial_Def.Reponse_Def <> '' THEN
	                "FC_Raz_Def"(#Transf.Dial_Def.Index_Defaut);
	                #Transf._TransfCommun.CommunGeneral._Etp := #Transf._TransfCommun.CommunGeneral._EtpMemo;
	                RETURN;
	            END_IF;
	        END_REGION Cyclique Attente Acquitement
	END_CASE;

END_FUNCTION

